	//udiFileNo:UDINT;
	udiNovRam_BufferIndex:UDINT;
	udiFile_Index:UDINT;
END_VAR
VAR_INST
	arrDataFromFile:ARRAY[0..GVL.arrArrayLength[E_DB_StructureType.SoDuration]-1] OF ST_SoDuration;//small
	DataToDB:ST_SoDuration;//large
	AnalizeIndex:UDINT;//should be kept by NovRam
	iStep:INT;
	i:UDINT;
	fbFileRingBuffer: FB_FileRingBuffer := ( sNetId     := '',
                                             sPathName  := '',
                                             ePath      := PATH_GENERIC,
                                             nID        := 1,
                                             cbBuffer   := gvl.arrFileRingBufferSize[E_DB_StructureType.ProductionSummary], //5MB(5*10^6Bytes)
                                             bOverwrite := FALSE,
                                             pWriteBuff := 0,
                                             cbWriteLen := 0,
                                             pReadBuff  := 0,
                                             cbReadLen  := 0,
                                             tTimeout   := T#1S );
	bBusy:BOOL;
	bError:BOOL;
	nErrID:UDINT;
	stHeader:ST_FileRBufferHead;
    //loadData  : ARRAY[0..511] OF BYTE :=[512(0)];
    //cbLoad    : UDINT;
	
	fileName: STRING(255);
	eStrIndex:DINT;
	fbSoDuration_DB:FB_SoDuration_DB;
	
END_VAR
//Config
eStrIndex:=E_DB_StructureType.SoDuration;

fbFileRingBuffer(sPathName:=fileName
				,bBusy=>bBusy,bError=>bError,nErrID=>nErrID
				,stHeader=>stHeader);
				
CASE iStep OF
	0://check if file full 
		IF NovRamData.arrFileRingBuffer_Status[eStrIndex].bFileFull[udiNovRam_BufferIndex][udiFile_Index] = TRUE//file full = should work 
		THEN
			
			fileName:=M_GetFileName(structureType:=eStrIndex
									,udiNovRam_BufferIndex:=udiNovRam_BufferIndex
									,udiFile_Index:=udiFile_Index);
			
			iStep:=100;
		END_IF
	100:// Open file
		
		AnalizeIndex:=0;
		fbFileRingBuffer.A_Open();
		
		iStep:=200;
	200://wait done / read head
		IF NOT fbFileRingBuffer.bBusy AND NOT fbFileRingBuffer.bError THEN
			
			fbFileRingBuffer.A_GetHead(pReadBuff := ADR(arrDataFromFile), cbReadLen := SIZEOF(arrDataFromFile));
			
			iStep:=300;
		END_IF
	300://wait done / take data from array
		IF NOT fbFileRingBuffer.bBusy AND NOT fbFileRingBuffer.bError THEN
			
			M_ST_SoDuration_Extract(Input:=arrDataFromFile[AnalizeIndex],Output=>DataToDB);
			//DataToDB:=arrDataFromFile[AnalizeIndex];
			
			iStep:=310;
		ELSIF NOT fbFileRingBuffer.bBusy AND fbFileRingBuffer.bError THEN//Empty
			iStep:=600;
		END_IF
	310:// write to DB
	
		IF fbSoDuration_DB.M_Upload(stSoDuration:=DataToDB) THEN
			iStep:=320;
		END_IF
		
	320://wait done
		
		IF NOT fbSoDuration_DB.bError THEN//write OK
		
			AnalizeIndex:=AnalizeIndex+1;
			
			iStep:=330;
			
		ELSE//write failed need to write to log
			;
		END_IF
		
	330://Check if all data in array Analized
		IF AnalizeIndex < GVL.arrArrayLength[eStrIndex]-1 THEN//not done
			iStep:=300;//go back
		ELSE//array data done
			iStep:=400;//complete this array
		END_IF
		
	400://wait done / remove Head
	
		fbFileRingBuffer.A_RemoveHead(pReadBuff := ADR(arrDataFromFile), cbReadLen := SIZEOF(arrDataFromFile));
		
		iStep:=500;
		
	500://wait done / check if all data got?
		IF NOT fbFileRingBuffer.bBusy AND NOT fbFileRingBuffer.bError THEN
			IF stHeader.nCount > 0 THEN
				iStep:=100;//Go Back
			ELSE
				iStep:=600;//finish
			END_IF
		END_IF
	600://reset file
	
		fbFileRingBuffer.A_Reset();
		
		iStep:=700;
		
	700://wait done / close file
		IF NOT fbFileRingBuffer.bBusy AND NOT fbFileRingBuffer.bError THEN
			
			fbFileRingBuffer.A_Close();
			
			iStep:=800;
		END_IF
	800://wait done
		IF NOT fbFileRingBuffer.bBusy AND NOT fbFileRingBuffer.bError THEN
			
			NovRamData.arrFileRingBuffer_Status[eStrIndex].bFileFull[udiNovRam_BufferIndex][udiFile_Index]:=FALSE;
			
			iStep:=0;
			
		END_IF
		
	
END_CASE
END_METHOD

METHOD M_ST_AlarmHistory_Extract : BOOL
VAR_INPUT
	Input:ST_AlarmInfo_DB_save;
END_VAR
VAR_OUTPUT
	Output:ST_AlarmInfo_DB;
END_VAR
Output.lrTime_ms:=Input.lrTime_ms;
Output.iMsgProc:=Input.iMsgProc;
Output.iStateAfter:=Input.iStateAfter;
Output.iMsgClass:=Input.iMsgClass;
Output.diMsgNumber:=Input.diMsgNumber;
Output.sTimeString:=Input.sTimeString;
Output.wsMsgText:=Input.wsMsgText;
Output.sPLC:=Input.sPLC;
Output.wsEquipment:=Input.wsEquipment;
Output.sFaam_id:=Input.sFaam_id;
END_METHOD

METHOD M_ST_ProductionHistory_Extract : BOOL
VAR_INPUT
	Input:ST_PHI_GroupData_DB;
END_VAR
VAR_OUTPUT
	Output:ST_PHI_GroupData_DB;
END_VAR
Output:=Input;
END_METHOD

METHOD M_ST_ProductionReport_Extract : BOOL
VAR_INPUT
	Input:ST_OEE_ProductionReport;
END_VAR
VAR_OUTPUT
	Output:ST_OEE_ProductionReport;
END_VAR
Output:=Input;
END_METHOD

METHOD M_ST_ProductionSummary_Extract : BOOL
VAR_INPUT
	Input:ST_OEE_ProductionSummary;
END_VAR
VAR_OUTPUT
	Output:ST_OEE_ProductionSummary;
END_VAR
Output:=Input;
END_METHOD

METHOD M_ST_RegularCheckResults_Extract : BOOL
VAR_INPUT
	Input:ST_RegularCheck_Results;
END_VAR
VAR_OUTPUT
	Output:ST_RegularCheck_Results;
END_VAR
(*
Output.diStation_number:=Input.diStation_number;
Output.diTrack_number:=Input.diTrack_number;
Output.dtStart_time:=Input.dtStart_time;

IF Input.eSensor = E_RegularCheckSensorResult.Pass THEN
	Output.bSensor:=TRUE;
ELSE
	Output.bSensor:=FALSE;
END_IF

IF Input.eCamera = E_RegularCheckSensorResult.Pass THEN
	Output.bCamera:=TRUE;
ELSE
	Output.bCamera:=FALSE;
END_IF

IF Input.eLoadcell = E_RegularCheckSensorResult.Pass THEN
	Output.bLoadcell:=TRUE;
ELSE
	Output.bLoadcell:=FALSE;
END_IF

IF Input.eSensor2 = E_RegularCheckSensorResult.Pass THEN
	Output.bSensor2:=TRUE;
ELSE
	Output.bSensor2:=FALSE;
END_IF

Output.diRegular_check_id:=Input.diRegular_check_id;
Output.sFaam_id:=Input.sFaam_id;
Output.sSo_number:=Input.sSo_number;
Output.diSo_id:=Input.diSo_id;
Output.wsEmployee_name_logged_in:=Input.wsEmployee_name_logged_in;
*)
Output:=Input;
END_METHOD

METHOD M_ST_SoDuration_Extract : BOOL
VAR_INPUT
	Input:ST_SoDuration;
END_VAR
VAR_OUTPUT
	Output:ST_SoDuration;
END_VAR
Output:=Input;
END_METHOD

METHOD M_ST_StopCount_Extract : BOOL
VAR_INPUT
	Input:ST_StopCount;
END_VAR
VAR_OUTPUT
	Output:ST_StopCount;
END_VAR
Output:=Input;
END_METHOD

METHOD M_StopCount : BOOL
VAR_INPUT
	
	//udiFileNo:UDINT;
	udiNovRam_BufferIndex:UDINT;
	udiFile_Index:UDINT;
END_VAR
VAR_INST
	arrDataFromFile:ARRAY[0..GVL.arrArrayLength[E_DB_StructureType.StopCount]-1] OF ST_StopCount;//small
	DataToDB:ST_StopCount;//large
	AnalizeIndex:UDINT;//should be kept by NovRam
	iStep:INT;
	i:UDINT;
	fbFileRingBuffer: FB_FileRingBuffer := ( sNetId     := '',
                                             sPathName  := '',
                                             ePath      := PATH_GENERIC,
                                             nID        := 1,
                                             cbBuffer   := gvl.arrFileRingBufferSize[E_DB_StructureType.StopCount], //5MB(5*10^6Bytes)
                                             bOverwrite := FALSE,
                                             pWriteBuff := 0,
                                             cbWriteLen := 0,
                                             pReadBuff  := 0,
                                             cbReadLen  := 0,
                                             tTimeout   := T#1S );
	bBusy:BOOL;
	bError:BOOL;
	nErrID:UDINT;
	stHeader:ST_FileRBufferHead;
    //loadData  : ARRAY[0..511] OF BYTE :=[512(0)];
    //cbLoad    : UDINT;
	
	fileName: STRING(255);
	eStrIndex:DINT;
	fbStopCount_DB:FB_StopCount_DB;
END_VAR
//Config
eStrIndex:=E_DB_StructureType.StopCount;

fbFileRingBuffer(sPathName:=fileName
				,bBusy=>bBusy,bError=>bError,nErrID=>nErrID
				,stHeader=>stHeader);
				
CASE iStep OF
	0://check if file full 
		IF NovRamData.arrFileRingBuffer_Status[eStrIndex].bFileFull[udiNovRam_BufferIndex][udiFile_Index] = TRUE//file full = should work 
		THEN
			
			fileName:=M_GetFileName(structureType:=eStrIndex
									,udiNovRam_BufferIndex:=udiNovRam_BufferIndex
									,udiFile_Index:=udiFile_Index);
			
			iStep:=100;
		END_IF
	100:// Open file
		
		AnalizeIndex:=0;
		fbFileRingBuffer.A_Open();
		
		iStep:=200;
	200://wait done / read head
		IF NOT fbFileRingBuffer.bBusy AND NOT fbFileRingBuffer.bError THEN
			
			fbFileRingBuffer.A_GetHead(pReadBuff := ADR(arrDataFromFile), cbReadLen := SIZEOF(arrDataFromFile));
			
			iStep:=300;
		END_IF
	300://wait done / take data from array
		IF NOT fbFileRingBuffer.bBusy AND NOT fbFileRingBuffer.bError THEN
			
			M_ST_StopCount_Extract(Input:=arrDataFromFile[AnalizeIndex],Output=>DataToDB);
			//DataToDB:=arrDataFromFile[AnalizeIndex];
			
			iStep:=310;
		ELSIF NOT fbFileRingBuffer.bBusy AND fbFileRingBuffer.bError THEN//Empty
			iStep:=600;
		END_IF
	310:// write to DB
		
		IF fbStopCount_DB.M_Upload(stStopCount:=DataToDB) THEN
			iStep:=320;
		END_IF
		
	320://wait done
		
		IF NOT fbStopCount_DB.bError THEN//write OK
		
			AnalizeIndex:=AnalizeIndex+1;
			
			iStep:=330;
			
		ELSE//write failed need to write to log
			;
		END_IF
		
	330://Check if all data in array Analized
		IF AnalizeIndex < GVL.arrArrayLength[eStrIndex]-1 THEN//not done
			iStep:=300;//go back
		ELSE//array data done
			iStep:=400;//complete this array
		END_IF
		
	400://wait done / remove Head
	
		fbFileRingBuffer.A_RemoveHead(pReadBuff := ADR(arrDataFromFile), cbReadLen := SIZEOF(arrDataFromFile));
		
		iStep:=500;
		
	500://wait done / check if all data got?
		IF NOT fbFileRingBuffer.bBusy AND NOT fbFileRingBuffer.bError THEN
			IF stHeader.nCount > 0 THEN
				iStep:=100;//Go Back
			ELSE
				iStep:=600;//finish
			END_IF
		END_IF
	600://reset file
	
		fbFileRingBuffer.A_Reset();
		
		iStep:=700;
		
	700://wait done / close file
		IF NOT fbFileRingBuffer.bBusy AND NOT fbFileRingBuffer.bError THEN
			
			fbFileRingBuffer.A_Close();
			
			iStep:=800;
		END_IF
	800://wait done
		IF NOT fbFileRingBuffer.bBusy AND NOT fbFileRingBuffer.bError THEN
			
			NovRamData.arrFileRingBuffer_Status[eStrIndex].bFileFull[udiNovRam_BufferIndex][udiFile_Index]:=FALSE;
			
			iStep:=0;
			
		END_IF
		
	
END_CASE
END_METHOD

END_FUNCTION_BLOCK

// ---- POUs/CheckBounds.TcPOU
// Implicitly generated code : DO NOT EDIT
FUNCTION CheckBounds : DINT
VAR_INPUT
	index, lower, upper: DINT;
END_VAR

// Implicitly generated code : Only an Implementation suggestion
{noflow}
IF  index < lower THEN
	GVL.udiLowerCnt := GVL.udiLowerCnt + 1;
	IF GVL.udiLowerCnt >= 1000000 THEN
		GVL.udiLowerCnt := 0;
	END_IF
	CheckBounds := lower;
ELSIF  index > upper THEN
	GVL.udiUpperCnt := GVL.udiUpperCnt + 1;
	IF GVL.udiUpperCnt >= 1000000 THEN
		GVL.udiUpperCnt := 0;
	END_IF
	CheckBounds := upper;
ELSE  
	CheckBounds := index;
END_IF
{flow}

END_FUNCTION
